// TIA Portal V19 export
FUNCTION "FC_FW_Auftrag_Step2_NB" : Void   // FC182, LAD
TITLE = Schritt CM03 -> CM01/CM02
{ S7_Optimized_Access := 'TRUE' }
// Ältesten Warenträger in CM03 suchen und nach CM01/CM02 transportieren
// stored: AutoNumber false, SetENOAutomatically false
   VAR_INPUT
      Frg_Schritt : Bool;
   END_VAR
   VAR_OUTPUT
      nextStep : Bool;
      startStep : Bool;
      parkStep : Bool;
   END_VAR
   VAR_IN_OUT
      Quelle : Int;
      Ziel : Int;
      Positionen : Array[1..30] of "UDT_Auftrag_Pos";
   END_VAR
   VAR_TEMP
      Sperre_Kurz_li : Bool;
      Sperre_Kurz_re : Bool;
      Sperre_Lang : Bool;
      Vorzug : Bool;
      Vorzug1 : Bool;
      Vorzug2 : Bool;
      Vorzug3 : Bool;
      Vorzug4 : Bool;
      Befehl_ok : Bool;
      tmpQuelle : Int;
      Oldest : Real;
   END_VAR
   VAR CONSTANT
      Wt_Cmd_Aetzen : Int := 1;
   END_VAR
BEGIN

REGION Network 1 (SCL)
   IF (#Quelle <> 0) AND (#Ziel <> 0) THEN
       #nextStep := #Positionen[#Quelle].Sperre;
       #startStep := NOT #nextStep;
       #Quelle := 0;
       #Ziel := 0;
       RETURN;
   END_IF;

   #Quelle := 0;
   #Ziel := 0;
   #nextStep := FALSE;
   #startStep := FALSE;

   IF NOT #Frg_Schritt THEN
       #nextStep := TRUE;
       RETURN;
   END_IF;
END_REGION

REGION Network 2 (SCL): Positionen sperren
   //Groß links nicht möglich
   #Positionen[9].CheckSperre := (#Positionen[3].Sperre AND #Positionen[15].Sperre) OR (#Positionen[9].Wt_Cmd <> #Wt_Cmd_Aetzen);

   //Groß rechts nicht möglich
   #Positionen[10].CheckSperre := (#Positionen[4].Sperre AND #Positionen[16].Sperre) OR (#Positionen[10].Wt_Cmd <> #Wt_Cmd_Aetzen);

   //kein Platz für Kurz links in CM01/CM02
   #Sperre_Kurz_li := #Positionen[1].Sperre AND #Positionen[5].Sperre AND #Positionen[13].Sperre AND #Positionen[17].Sperre;

   //kein Platz für Kurz rechts in CM01/CM02
   #Sperre_Kurz_re := #Positionen[2].Sperre AND #Positionen[6].Sperre AND #Positionen[14].Sperre AND #Positionen[18].Sperre;

   //kein Platz für Lang in CM01/CM02
   #Sperre_Lang := (#Positionen[1].Sperre OR #Positionen[2].Sperre) AND (#Positionen[5].Sperre OR #Positionen[6].Sperre) AND (#Positionen[13].Sperre OR #Positionen[14].Sperre) AND (#Positionen[17].Sperre OR #Positionen[18].Sperre);

   //Lang in P7 oder
   //kein Platz auf rechter Seite
   //-> P8 sperren
   #Positionen[8].CheckSperre := #Sperre_Kurz_re OR (#Positionen[7].Wt_Typ = "WT_Typ_LS") OR (#Positionen[8].Wt_Cmd <> #Wt_Cmd_Aetzen);

   //Lang in P7 und kein Platz für Lang oder
   //kein Platz auf linker Seite
   //-> P7 sperren
   #Positionen[7].CheckSperre := #Sperre_Kurz_li OR ((#Positionen[7].Wt_Typ = "WT_Typ_LS") AND #Sperre_Lang) OR (#Positionen[7].Wt_Cmd <> #Wt_Cmd_Aetzen);

   //Lang in P11 oder
   //kein Platz auf rechter Seite
   //-> P12 sperren
   #Positionen[12].CheckSperre := #Sperre_Kurz_re OR (#Positionen[11].Wt_Typ = "WT_Typ_LS") OR (#Positionen[12].Wt_Cmd <> #Wt_Cmd_Aetzen);

   //Lang in P11 und kein Platz für Lang oder
   //kein Platz auf linker Seite
   //-> P11 sperren
   #Positionen[11].CheckSperre := #Sperre_Kurz_li OR ((#Positionen[11].Wt_Typ = "WT_Typ_LS") AND #Sperre_Lang) OR (#Positionen[11].Wt_Cmd <> #Wt_Cmd_Aetzen);
END_REGION

REGION Network 3 (SCL): Ältesten WT suchen
   //
   #Oldest := 0;
   #tmpQuelle := 0;

   //CM03
   "FC_FW_Auftrag_Suche"(Pos1 := 7,
                         Pos2 := 12,
                         Positionen := #Positionen,
                         Quelle := #tmpQuelle,
                         Oldest := #Oldest);
END_REGION

REGION Network 4 (SCL): Auswertung
   IF #tmpQuelle = 0 THEN
       //kein WT
       #nextStep := TRUE;
       RETURN;
   END_IF;

   IF NOT #Positionen[#tmpQuelle].Fertig THEN
       #parkStep := TRUE;
       RETURN;
   END_IF;

   IF (#tmpQuelle = 9) THEN
       //Gross links
       IF NOT #Positionen[3].Sperre THEN
           "FC_FW_Auftrag_Befehl"(inQuelle := #tmpQuelle,
                                  inZiel := 3,
                                  Befehl_ok => #Befehl_ok,
                                  outQuelle => #Quelle,
                                  outZiel => #Ziel);

           #nextStep := NOT #Befehl_ok;
       ELSIF NOT #Positionen[15].Sperre THEN
           "FC_FW_Auftrag_Befehl"(inQuelle := #tmpQuelle,
                                  inZiel := 15,
                                  Befehl_ok => #Befehl_ok,
                                  outQuelle => #Quelle,
                                  outZiel => #Ziel);

           #nextStep := NOT #Befehl_ok;
       ELSE
           #nextStep := TRUE;
       END_IF;
       RETURN;
   END_IF;

   IF (#tmpQuelle = 10) THEN
       //Gross rechts
       IF NOT #Positionen[4].Sperre THEN
           "FC_FW_Auftrag_Befehl"(inQuelle := #tmpQuelle,
                                  inZiel := 4,
                                  Befehl_ok => #Befehl_ok,
                                  outQuelle => #Quelle,
                                  outZiel => #Ziel);

           #nextStep := NOT #Befehl_ok;
       ELSIF NOT #Positionen[16].Sperre THEN
           "FC_FW_Auftrag_Befehl"(inQuelle := #tmpQuelle,
                                  inZiel := 16,
                                  Befehl_ok => #Befehl_ok,
                                  outQuelle => #Quelle,
                                  outZiel => #Ziel);

           #nextStep := NOT #Befehl_ok;
       ELSE
           #nextStep := TRUE;
       END_IF;
       RETURN;
   END_IF;

   IF (#Positionen[#tmpQuelle].Wt_Typ = "WT_Typ_LS") AND ((#tmpQuelle = 7) OR (#tmpQuelle = 11)) THEN
       //Lang
       IF NOT #Positionen[13].Sperre AND NOT #Positionen[14].Sperre THEN
           "FC_FW_Auftrag_Befehl"(inQuelle := #tmpQuelle,
                                  inZiel := 13,
                                  Befehl_ok => #Befehl_ok,
                                  outQuelle => #Quelle,
                                  outZiel => #Ziel);

           #nextStep := NOT #Befehl_ok;
       ELSIF NOT #Positionen[5].Sperre AND NOT #Positionen[6].Sperre THEN
           "FC_FW_Auftrag_Befehl"(inQuelle := #tmpQuelle,
                                  inZiel := 5,
                                  Befehl_ok => #Befehl_ok,
                                  outQuelle => #Quelle,
                                  outZiel => #Ziel);

           #nextStep := NOT #Befehl_ok;
       ELSIF NOT #Positionen[1].Sperre AND NOT #Positionen[2].Sperre THEN
           "FC_FW_Auftrag_Befehl"(inQuelle := #tmpQuelle,
                                  inZiel := 1,
                                  Befehl_ok => #Befehl_ok,
                                  outQuelle => #Quelle,
                                  outZiel => #Ziel);

           #nextStep := NOT #Befehl_ok;
       ELSIF NOT #Positionen[17].Sperre AND NOT #Positionen[18].Sperre THEN
           "FC_FW_Auftrag_Befehl"(inQuelle := #tmpQuelle,
                                  inZiel := 17,
                                  Befehl_ok => #Befehl_ok,
                                  outQuelle => #Quelle,
                                  outZiel => #Ziel);

           #nextStep := NOT #Befehl_ok;
       ELSE
           #nextStep := TRUE;
       END_IF;
       RETURN;
   END_IF;

   IF (#tmpQuelle = 7) OR (#tmpQuelle = 11) THEN
       //Kurz links
       #Vorzug1 := NOT #Positionen[1].Sperre AND #Positionen[2].Sperre;
       #Vorzug2 := NOT #Positionen[5].Sperre AND #Positionen[6].Sperre;
       #Vorzug3 := NOT #Positionen[13].Sperre AND #Positionen[14].Sperre;
       #Vorzug4 := NOT #Positionen[17].Sperre AND #Positionen[18].Sperre;

       #Vorzug := NOT #Vorzug2 AND (#Vorzug1 OR #Vorzug3 OR #Vorzug4);
       IF NOT #Positionen[5].Sperre AND NOT #Vorzug THEN
           "FC_FW_Auftrag_Befehl"(inQuelle := #tmpQuelle,
                                  inZiel := 5,
                                  Befehl_ok => #Befehl_ok,
                                  outQuelle => #Quelle,
                                  outZiel => #Ziel);

           #nextStep := NOT #Befehl_ok;
           RETURN;
       END_IF;

       #Vorzug := NOT #Vorzug3 AND (#Vorzug1 OR #Vorzug4);
       IF NOT #Positionen[13].Sperre AND NOT #Vorzug THEN
           "FC_FW_Auftrag_Befehl"(inQuelle := #tmpQuelle,
                                  inZiel := 13,
                                  Befehl_ok => #Befehl_ok,
                                  outQuelle => #Quelle,
                                  outZiel => #Ziel);

           #nextStep := NOT #Befehl_ok;
           RETURN;
       END_IF;

       #Vorzug := NOT #Vorzug1 AND #Vorzug4;
       IF NOT #Positionen[1].Sperre AND NOT #Vorzug THEN
           "FC_FW_Auftrag_Befehl"(inQuelle := #tmpQuelle,
                                  inZiel := 1,
                                  Befehl_ok => #Befehl_ok,
                                  outQuelle => #Quelle,
                                  outZiel => #Ziel);

           #nextStep := NOT #Befehl_ok;
           RETURN;
       END_IF;

       IF NOT #Positionen[17].Sperre THEN
           "FC_FW_Auftrag_Befehl"(inQuelle := #tmpQuelle,
                                  inZiel := 17,
                                  Befehl_ok => #Befehl_ok,
                                  outQuelle => #Quelle,
                                  outZiel => #Ziel);

           #nextStep := NOT #Befehl_ok;
           RETURN;
       END_IF;

       #nextStep := TRUE;
       RETURN;
   END_IF;

   IF (#tmpQuelle = 8) OR (#tmpQuelle = 12) THEN
       //Kurz rechts
       #Vorzug1 := NOT #Positionen[2].Sperre AND #Positionen[1].Sperre;
       #Vorzug2 := NOT #Positionen[6].Sperre AND #Positionen[5].Sperre;
       #Vorzug3 := NOT #Positionen[14].Sperre AND #Positionen[13].Sperre;
       #Vorzug4 := NOT #Positionen[18].Sperre AND #Positionen[17].Sperre;

       #Vorzug := NOT #Vorzug2 AND (#Vorzug1 OR #Vorzug3 OR #Vorzug4);
       IF NOT #Positionen[6].Sperre AND NOT #Vorzug THEN
           "FC_FW_Auftrag_Befehl"(inQuelle := #tmpQuelle,
                                  inZiel := 6,
                                  Befehl_ok => #Befehl_ok,
                                  outQuelle => #Quelle,
                                  outZiel => #Ziel);

           #nextStep := NOT #Befehl_ok;
           RETURN;
       END_IF;

       #Vorzug := NOT #Vorzug3 AND (#Vorzug1 OR #Vorzug4);
       IF NOT #Positionen[14].Sperre AND NOT #Vorzug THEN
           "FC_FW_Auftrag_Befehl"(inQuelle := #tmpQuelle,
                                  inZiel := 14,
                                  Befehl_ok => #Befehl_ok,
                                  outQuelle => #Quelle,
                                  outZiel => #Ziel);

           #nextStep := NOT #Befehl_ok;
           RETURN;
       END_IF;

       #Vorzug := NOT #Vorzug1 AND #Vorzug4;
       IF NOT #Positionen[2].Sperre AND NOT #Vorzug THEN
           "FC_FW_Auftrag_Befehl"(inQuelle := #tmpQuelle,
                                  inZiel := 2,
                                  Befehl_ok => #Befehl_ok,
                                  outQuelle => #Quelle,
                                  outZiel => #Ziel);

           #nextStep := NOT #Befehl_ok;
           RETURN;
       END_IF;

       IF NOT #Positionen[18].Sperre THEN
           "FC_FW_Auftrag_Befehl"(inQuelle := #tmpQuelle,
                                  inZiel := 18,
                                  Befehl_ok => #Befehl_ok,
                                  outQuelle => #Quelle,
                                  outZiel => #Ziel);

           #nextStep := NOT #Befehl_ok;
           RETURN;
       END_IF;

       #nextStep := TRUE;
       RETURN;
   END_IF;

   //?
   #nextStep := TRUE;
END_REGION
END_FUNCTION
